ABB RobotStudio station: Practica5Avanzada_EstacionDePartida_1.rspag

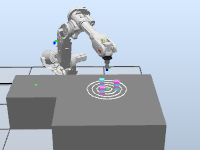
--- station ---
Station Practica3Avanzada_EstacionDePartida_1 (saved by RobotStudio 20.4.9280.0)
Controller Sistema6
  mechanical unit ROB_1: IRB6640_180_255__04, 6 joints, base frame (0, 0, 0) mm
Layout (positions relative to the parent item):
  - Ventosa [mechanism] at (1700, 1000, 1450) mm, rotated rx -180 ry 0 rz -180 deg
      TCP Ventosa at (0, 0, 200) mm
      links: PiezaVentosa
  - IRB6640_180_255__04 [mechanism, from Robots\IRB6640_180_255_G_04.rslib] at (0, 0, 0) mm; joint values [0.5317, 0.479, -0.2332, 0, 1.325, 0.5317] (rad or m)
  - MesaTrabajoParte1 [part]
  - MesaTrabajoParte0 [part]
  - CI_VentosaVacuostato [smart component]
      signals: DI ActivaVentosa, DO Vacuostato
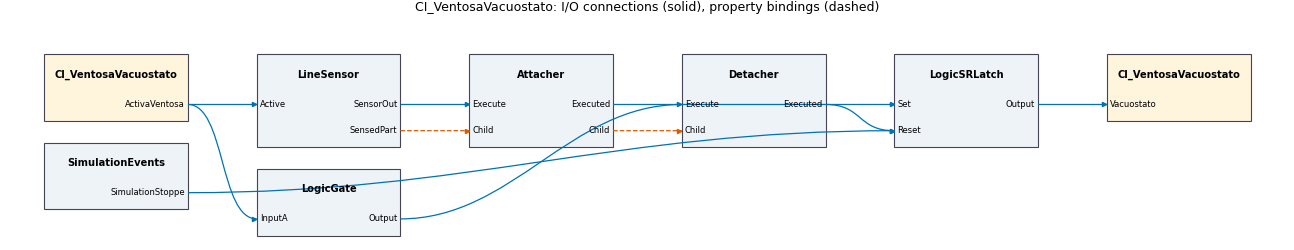
      connections:
        CI_VentosaVacuostato.ActivaVentosa -> LineSensor.Active
        LineSensor.SensorOut -> Attacher.Execute
        Attacher.Executed -> LogicSRLatch.Set
        LogicSRLatch.Output -> CI_VentosaVacuostato.Vacuostato
        Detacher.Executed -> LogicSRLatch.Reset
        SimulationEvents.SimulationStopped -> LogicSRLatch.Reset
        CI_VentosaVacuostato.ActivaVentosa -> LogicGate.InputA
        LogicGate.Output -> Detacher.Execute
        LineSensor.SensedPart => Attacher.Child
        Attacher.Child => Detacher.Child
    - LineSensor [smart component, from Components\LineSensor.rslib] at (1700, 1000, 1250) mm, rotated rx -180 ry 0 rz -180 deg
        properties: Start=[0 0 -0.002]; End=[0 0 0.02]; Radius=0.002; SensedPart=Pieza1; SensedPoint=[1.7 1.2 0.950000061035156]
      - _sensorPart_ [part]
    - SimulationEvents [smart component, from Components\SimulationEvents.rslib]
    - LogicSRLatch [smart component, from Components\LogicSRLatch.rslib]
    - Attacher [smart component, from Components\Attacher.rslib]
        properties: Parent=Ventosa; Flange=0; Child=Pieza1; Mount=false; Offset=[0 0 0]; Orientation=[0 0 0]
    - Detacher [smart component, from Components\Detacher.rslib]
        properties: Child=Pieza1; KeepPosition=true
    - LogicGate [smart component, from Components\LogicGate.rslib]
        properties: Operator=NOT; Delay=0.1
  - MesaTrabajoParte2 [part] at (0, 1000, 0) mm
  - MesaTrabajoParte3 [part] at (1000, 0, 0) mm
  - MesaTrabajoParte4 [part] at (1000, 1000, 0) mm
  - Pieza1 [part] at (200, 1700, 150) mm
  - Pieza2 [part] at (26.79, 1400, 50) mm
  - Pieza3 [part] at (373.21, 1400, 0) mm
  - Pieza4 [part] at (200, 1700, -50) mm
  - Pieza5 [part] at (26.79, 1400, -150) mm
  - CircunferenciaR200 [part]
  - CircunferenciaR100 [part]
  - CircunferenciaR300 [part]
  - CircunferenciaR400 [part]
  - Pieza6 [part] at (373.21, 1400, -200) mm
  - Pieza7 [part] at (200, 1700, -250) mm
  - Pieza8 [part] at (26.79, 1400, -350) mm
  - Pieza9 [part] at (373.2, 1400, -400) mm
  - Pieza10 [part] at (200, 1700, -450) mm
Attachment: LineSensor is attached to Ventosa / PiezaVentosa
Attachment: Ventosa is attached to IRB6640_180_255__04 / Link6
Station logic (signal -> signal, property => property):
  CI_VentosaVacuostato.Vacuostato -> Sistema6.ED_PiezaCogida
  Sistema6.SD_ActivaVentosa -> CI_VentosaVacuostato.ActivaVentosa

--- Backups/Sistema6/RAPID/TASK1/PROGMOD/CalibData.mod ---
MODULE CalibData
	PERS tooldata Ventosa:=[TRUE,[[0,0,200],[1,0,0,0]],[1,[0,0,125],[1,0,0,0],0.002,0.002,0.0013]];
ENDMODULE

--- Backups/Sistema6/RAPID/TASK1/PROGMOD/Module1.mod ---
MODULE Module1
    CONST robtarget pBaseOrigen:=[[1500,-500,750],[0,0,1,0],[0,0,0,0],[9E+09,9E+09,9E+09,9E+09,9E+09,9E+09]];
    CONST robtarget pCentroDestino:=[[1700,1000,750],[0,0,1,0],[0,0,0,0],[9E+09,9E+09,9E+09,9E+09,9E+09,9E+09]];
    CONST robtarget pReposo:=[[1808.910161514,0,1855],[0.5,0,0.866025404,0],[0,0,0,0],[9E+09,9E+09,9E+09,9E+09,9E+09,9E+09]];

    !Constantes creadas por mi
    CONST num altura := 50;
    CONST num numeroDeTorresDestino := 3;
    CONST num nPiezasEnElOrigen := 10;

    PROC main()
        Ejercicio2 10, numeroDeTorresDestino, 200;
    ENDPROC

    PROC Ejercicio2 (num nPiezasTorreOrigen, num nTorresDestino, num radioCircunferencia)
        VAR robtarget tabPos{numeroDeTorresDestino};
        VAR robtarget pAproxCirculo;
        VAR robtarget pAproxOrigen;
        VAR robtarget pBase;
        VAR robtarget pAux;
        VAR robtarget pApoyo;
        VAR num gradosIncremt := 0;
        VAR num grados := 0;
        VAR num nPiezasEnTorre := 0;
        VAR num alturaTorreDestino := 0;
        VAR num alturaTorreOrigen := 0;
        VAR num X := 0;
        VAR num Y := 0;
        VAR num hipotenusa;

        !Inicializamos
        alturaTorreOrigen := altura * nPiezasTorreOrigen;

        !Vamos a crear un punto de aproximación encima del centro del circulo y 5 piezas por encima de la torre origen
        pAproxCirculo := Offs (pCentroDestino, 0, 0, altura * nPiezasTorreOrigen);
        pAproxOrigen := Offs (pBaseOrigen, 0, 0, (nPiezasTorreOrigen * altura) + (altura * 5));

        !Creamos el punto inicial de la torre origen
        pBase := Offs (pBaseOrigen, 0, 0, altura * nPiezasTorreOrigen);

        !Como el círculo tiene 360 grados, podemos descomponen los grados en tantas partes como puntos tenemos
        gradosIncremt := 360 / nTorresDestino;
        alturaTorreDestino := altura;
        hipotenusa := radioCircunferencia;

        !Vamos a buscar las posiciones de las torres destino
        FOR i FROM 1 TO nTorresDestino DO

            !Calculamos las posiciones haciendo uso de senos y cosenos
            X := Sin(grados) * hipotenusa;
            Y := Cos(grados) * hipotenusa;

            !Creamos los puntos
            pAux := Offs (pCentroDestino, X, Y, 0);

            !Lo añadimos en la tabla
            tabPos{i} := pAux;

            !Actualizamos los grados
            grados := grados + gradosIncremt;

        ENDFOR

        !En este segundo bucle for recorremos todos los puntos del array cogiendo y dejando las piezas
        FOR A FROM 1 TO nPiezasTorreOrigen DO
            FOR B FROM 1 TO nTorresDestino DO

                !Restriccion para que una vez se acaben las piezas no haga nada
                IF alturaTorreOrigen <= 0 THEN
                    Break;
                ELSE

                !Movemos al punto de aproximación de la Torre Origen
                MoveL pAproxOrigen, v2000, fine, Ventosa\WObj:=wobj0;

                !Cogemos la pieza de la Torre Origen
                MoveLDO pBase, v2000, fine, Ventosa\WObj:=wobj0, SD_ActivaVentosa, 1;
                WaitDI ED_PiezaCogida, 1;
                MoveL pAproxOrigen, v2000, fine, Ventosa\WObj:=wobj0;

                !Movemos al punto de aproximacion del centro del círculo;
                MoveL pAproxCirculo, v2000, fine, Ventosa\WObj:=wobj0;

                !Depositamos la pieza en su sitio
                pApoyo := Offs (tabPos{B}, 0, 0, alturaTorreDestino);
                MoveLDO pApoyo, v2000, fine, Ventosa\WObj:=wobj0, SD_ActivaVentosa, 0;
                WaitDI ED_PiezaCogida, 0;
                MoveL pAproxCirculo, v2000, fine, Ventosa\WObj:=wobj0;

                !Bajamos la altura de la torre Base
                pBase := Offs (pBase, 0, 0, -altura);

                ENDIF

                !Decrementamos la altura en la torre origen para poder usar la restricción de altura
                alturaTorreOrigen := alturaTorreOrigen - altura;

            ENDFOR

            !Cuando colocamos todas las torres con la misma altura la actualizamos
            alturaTorreDestino := alturaTorreDestino + altura;

        ENDFOR

    ENDPROC

ENDMODULE

--- Backups/Sistema6/RAPID/TASK1/SYSMOD/LINKEDM.sys ---
%%%
  VERSION:1
  LANGUAGE:ENGLISH
%%%

MODULE LINKEDM (SYSMODULE)

! FOLLOWER
!     Name of electronically linked follower axis used by operator at teach pendent.
      PERS string l_f_axis_name{5}       :=  ["",  "", "", "", ""];

!     Name of the mechanical unit for follower axis.
      PERS string l_f_mecunt_n{5}  :=  ["", "", "", "", ""];

!     Linked follower axis number in the mechanical unit (first axis in mech. unit is number 1).
      PERS num l_f_axis_no{5}      :=  [0,          0,   0,  0,  0];

! MASTER
!     Name of the mechanical unit for linked master axis.
      PERS string l_m_mecunt_n{5} :=  ["", "", "", "", ""];

!     Linked master axis number in the mechanical unit (first axis in mech. unit is number 1).
!     See axis number table in documentation for different master mechanical units.
      PERS num l_m_axis_no{5}     :=  [0,  0,  0,  0,  0];

! POSITION OFFSET
!     The increase of the allowed offset position between the master and follower
!     positions, used when starting AUTO mode. As soon as the offset is decreased
!     the old configurated parameter is used.
!     Example: 3 => the configurated value of allowed offset is increased 3 times.
      PERS num offset_ratio{5}       :=  [10,  10,   10,  10,  10];

! SPEED RATIO
!     Speed_ratio used in AUTO and JOG modes [ very_slow   slow    normal    fast]
!     Value 1 = max allowed manual speed.
      CONST num speed_ratio {20}      := [0.01, 0.01, 0.01, 0.01, 0.01,
                                          0.05, 0.05, 0.05, 0.05, 0.05,
                                          0.20, 0.20, 0.20, 0.20, 0.20,
                                          1.00, 1.00, 1.00, 1.00, 1.00];

! STEP SIZE
!     Displacement position used in JOG mode for each activation of positive or
!     negative movement.                  [very_short    short   normal   long]
!     Unit degees or meter.
      CONST num displacement {20}     := [0.001, 0.001, 0.001, 0.001, 0.001,
                                          0.005, 0.005, 0.005, 0.005, 0.005,
                                          0.020, 0.020, 0.020, 0.020, 0.020,
                                          0.100, 0.100, 0.100, 0.100, 0.100];


!-------------------------------------------------------------
 PROC Linked_m ()
      Linked_m_exe ;
 ENDPROC
ENDMODULE

--- Backups/Sistema6/SYSPAR/EIO.cfg ---
EIO:CFG_1.0:6:1::
#
INDUSTRIAL_NETWORK:

      -Name "DeviceNet" -Label "DeviceNet Master/Slave Network" -Address "2"
#
DEVICENET_DEVICE:

      -Name "MiDeviceNet" -Label "MiDeviceNet"
#
DEVICENET_INTERNAL_DEVICE:

      -Name "DN_Internal_Device" -VendorName "ABB Robotics"\
      -ProductName "DeviceNet Internal Slave Device"
#
EIO_SIGNAL:

      -Name "ED_PiezaCogida" -SignalType "DI" -Device "MiDeviceNet"\
      -Label "ED_PiezaCogida" -DeviceMap "0" -Access "All"

      -Name "SD_ActivaVentosa" -SignalType "DO" -Device "MiDeviceNet"\
      -Label "SD_ActivaVentosa" -DeviceMap "0" -Access "All"
